FUNCTION F_BuildJSON : STRING(255)
VAR_INPUT
	  Sensor1 : STRING(255);
	  Sensor2 : STRING(255);
	  Sensor3 : STRING(255);
END_VAR
VAR
	  sReturnValue : STRING(255);
END_VAR

sReturnValue := CONCAT('{ "Sensor1" : ', Sensor1);
sReturnValue := CONCAT(sReturnValue, ', "Sensor2" : ');
sReturnValue := CONCAT(sReturnValue, Sensor2);
sReturnValue := CONCAT(sReturnValue, ', "Sensor3" : ');
sReturnValue := CONCAT(sReturnValue, Sensor3);
sReturnValue := CONCAT(sReturnValue, '}');
F_BuildJSON := sReturnValue;

END_FUNCTION

(* stored: Version 1.1.0.1, ProductVersion 3.1.4021.12
   POU F_BuildJSON: Id {272d0e97-05c8-43c5-9509-dd91bc2a6f4e}, SpecialFunc None *)
